FUNCTION F_FindAddr : POINTER TO BYTE
VAR_INPUT
	pAddrTo: POINTER TO BYTE;
	nByteCount: UINT;
END_VAR
VAR

END_VAR

IF nByteCount=8 THEN
	pAddrTo := pAddrTo;
	nByteCount := 0;
ELSIF nByteCount>8 THEN
	pAddrTo := pAddrTo + 16 - nByteCount;
	nByteCount := 0;
ELSE
	pAddrTo := pAddrTo;
END_IF

F_FindAddr := pAddrTo;

END_FUNCTION

(* stored: Version 1.1.0.1, ProductVersion 3.1.4020.12
   POU F_FindAddr: Id {6257a32b-62d9-4df0-b406-77555b3d6a65}, SpecialFunc None *)
